// TIA Portal project "Parking_Lort_V15.1" (V15.1)

(* hardware
DEVICE "S7-1200 station_1"  S7-1200 Station
   slot 0: "Rack_0"  S7-1200 Rack  Rack  V1.0
   slot 1: "PLC_1"  CPU 1212C DC/DC/Rly  6ES7 212-1HE40-0XB0  V4.2
*)

// ===== PLC "PLC_1"  CPU 1212C DC/DC/Rly =====

VAR_GLOBAL   // PLC tag table "Default tag table"
   "I_IN barrier is down" AT %I0.0 : Bool;
   "I_IN barrier is up" AT %I0.1 : Bool;
   "I_OUT barrier is down" AT %I0.2 : Bool;
   "I_OUT barrier is up" AT %I0.3 : Bool;
   "I_Car is at the barrier IN" AT %I0.4 : Bool;
   "I_Car is at the barrier OUT" AT %I0.5 : Bool;
   "Q_IN barrier up" AT %Q0.0 : Bool;
   "Q_OUT barrier up" AT %Q0.1 : Bool;
   "Q_Red signal IN" AT %Q0.2 : Bool;
   "Q_Green signal IN" AT %Q0.3 : Bool;
   "Q_Red signal OUT" AT %Q0.4 : Bool;
   "Q_Green signal OUT" AT %Q0.5 : Bool;
END_VAR

DATA_BLOCK "Barrier_DB"   // DB1
{ S7_Optimized_Access := 'TRUE' }
VERSION : 0.1
// stored: InstanceOfName ENTER_Barrier
"ENTER_Barrier"
BEGIN
END_DATA_BLOCK

DATA_BLOCK "EXIT_Barrier_DB"   // DB2
{ S7_Optimized_Access := 'TRUE' }
VERSION : 0.1
// stored: InstanceOfName EXIT_Barrier
"EXIT_Barrier"
BEGIN
END_DATA_BLOCK

FUNCTION_BLOCK "ENTER_Barrier"   // FB1, LAD
TITLE = Barriers
{ S7_Optimized_Access := 'TRUE' }
VERSION : 0.1
BEGIN

REGION Network 1: ENTER
   // Condition to lift up the barrier
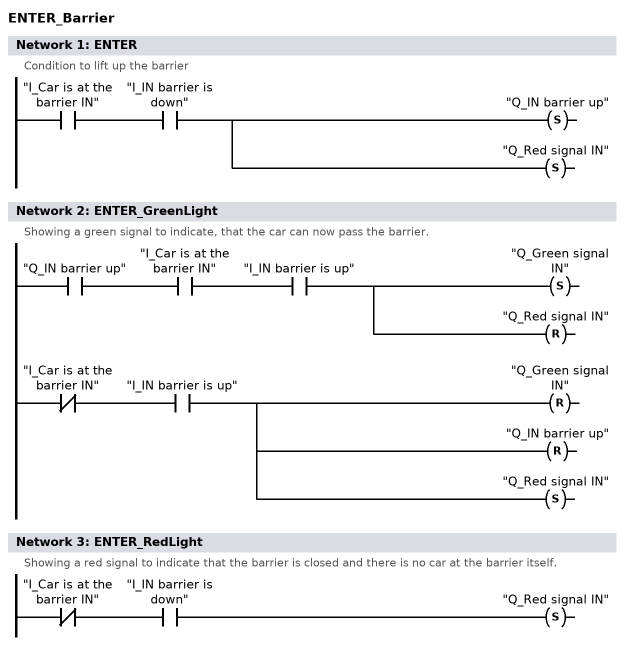
   RUNG wire#powerrail
      Contact( "I_Car is at the barrier IN" )
      Contact( "I_IN barrier is down" )
      wire#w1
      S_Coil( "Q_IN barrier up" )
   END_RUNG
   RUNG wire#w1
      S_Coil( "Q_Red signal IN" )
   END_RUNG
   // the same network as SCL:
   IF "I_Car is at the barrier IN" AND "I_IN barrier is down" THEN
       "Q_IN barrier up" := TRUE;
       "Q_Red signal IN" := TRUE;
   END_IF;
END_REGION

REGION Network 2: ENTER_GreenLight
   // Showing a green signal to indicate, that the car can now pass the barrier.
   RUNG wire#powerrail
      Contact( "Q_IN barrier up" )
      Contact( "I_Car is at the barrier IN" )
      Contact( "I_IN barrier is up" )
      wire#w1
      S_Coil( "Q_Green signal IN" )
   END_RUNG
   RUNG wire#w1
      R_Coil( "Q_Red signal IN" )
   END_RUNG
   RUNG wire#powerrail
      I_Contact( "I_Car is at the barrier IN" )
      Contact( "I_IN barrier is up" )
      wire#w2
      R_Coil( "Q_Green signal IN" )
   END_RUNG
   RUNG wire#w2
      R_Coil( "Q_IN barrier up" )
   END_RUNG
   RUNG wire#w2
      S_Coil( "Q_Red signal IN" )
   END_RUNG
   // the same network as SCL:
   IF "Q_IN barrier up" AND "I_Car is at the barrier IN" AND "I_IN barrier is up" THEN
       "Q_Green signal IN" := TRUE;
       "Q_Red signal IN" := FALSE;
   END_IF;
   IF NOT "I_Car is at the barrier IN" AND "I_IN barrier is up" THEN
       "Q_Green signal IN" := FALSE;
       "Q_IN barrier up" := FALSE;
       "Q_Red signal IN" := TRUE;
   END_IF;
END_REGION

REGION Network 3: ENTER_RedLight
   // Showing a red signal to indicate that the barrier is closed and there is no car at the barrier itself.
   RUNG wire#powerrail
      I_Contact( "I_Car is at the barrier IN" )
      Contact( "I_IN barrier is down" )
      S_Coil( "Q_Red signal IN" )
   END_RUNG
   // the same network as SCL:
   IF NOT "I_Car is at the barrier IN" AND "I_IN barrier is down" THEN "Q_Red signal IN" := TRUE; END_IF;
END_REGION
END_FUNCTION_BLOCK

FUNCTION_BLOCK "EXIT_Barrier"   // FB2, LAD
{ S7_Optimized_Access := 'TRUE' }
VERSION : 0.1
BEGIN

REGION Network 1: ENTER
   // Condition to lift up the barrier
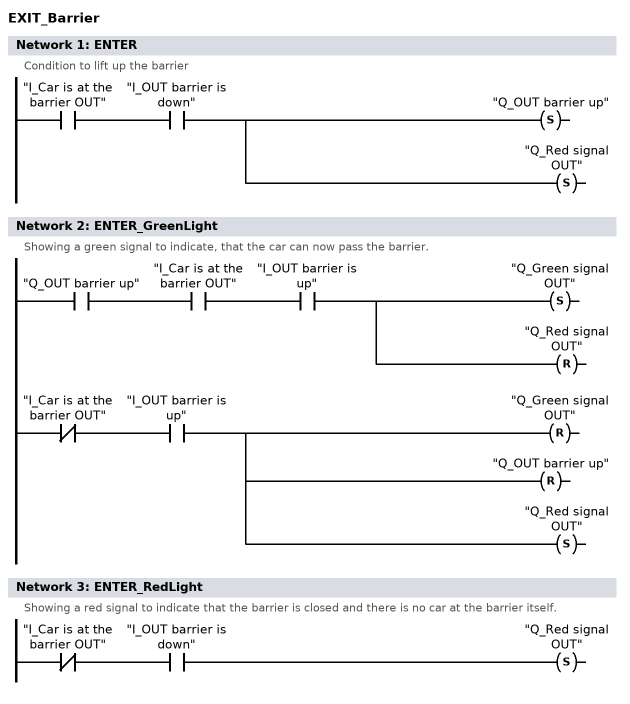
   RUNG wire#powerrail
      Contact( "I_Car is at the barrier OUT" )
      Contact( "I_OUT barrier is down" )
      wire#w1
      S_Coil( "Q_OUT barrier up" )
   END_RUNG
   RUNG wire#w1
      S_Coil( "Q_Red signal OUT" )
   END_RUNG
   // the same network as SCL:
   IF "I_Car is at the barrier OUT" AND "I_OUT barrier is down" THEN
       "Q_OUT barrier up" := TRUE;
       "Q_Red signal OUT" := TRUE;
   END_IF;
END_REGION

REGION Network 2: ENTER_GreenLight
   // Showing a green signal to indicate, that the car can now pass the barrier.
   RUNG wire#powerrail
      Contact( "Q_OUT barrier up" )
      Contact( "I_Car is at the barrier OUT" )
      Contact( "I_OUT barrier is up" )
      wire#w1
      S_Coil( "Q_Green signal OUT" )
   END_RUNG
   RUNG wire#w1
      R_Coil( "Q_Red signal OUT" )
   END_RUNG
   RUNG wire#powerrail
      I_Contact( "I_Car is at the barrier OUT" )
      Contact( "I_OUT barrier is up" )
      wire#w2
      R_Coil( "Q_Green signal OUT" )
   END_RUNG
   RUNG wire#w2
      R_Coil( "Q_OUT barrier up" )
   END_RUNG
   RUNG wire#w2
      S_Coil( "Q_Red signal OUT" )
   END_RUNG
   // the same network as SCL:
   IF "Q_OUT barrier up" AND "I_Car is at the barrier OUT" AND "I_OUT barrier is up" THEN
       "Q_Green signal OUT" := TRUE;
       "Q_Red signal OUT" := FALSE;
   END_IF;
   IF NOT "I_Car is at the barrier OUT" AND "I_OUT barrier is up" THEN
       "Q_Green signal OUT" := FALSE;
       "Q_OUT barrier up" := FALSE;
       "Q_Red signal OUT" := TRUE;
   END_IF;
END_REGION

REGION Network 3: ENTER_RedLight
   // Showing a red signal to indicate that the barrier is closed and there is no car at the barrier itself.
   RUNG wire#powerrail
      I_Contact( "I_Car is at the barrier OUT" )
      Contact( "I_OUT barrier is down" )
      S_Coil( "Q_Red signal OUT" )
   END_RUNG
   // the same network as SCL:
   IF NOT "I_Car is at the barrier OUT" AND "I_OUT barrier is down" THEN "Q_Red signal OUT" := TRUE; END_IF;
END_REGION
END_FUNCTION_BLOCK

ORGANIZATION_BLOCK "Main"   // OB1, LAD, ProgramCycle
TITLE = "Main Program Sweep (Cycle)"
{ S7_Optimized_Access := 'TRUE' }
VERSION : 0.1
   VAR_INPUT
      Initial_Call : Bool;   // Initial call of this OB
      Remanence : Bool;   // =True, if remanent data are available
   END_VAR
BEGIN

REGION Network 1
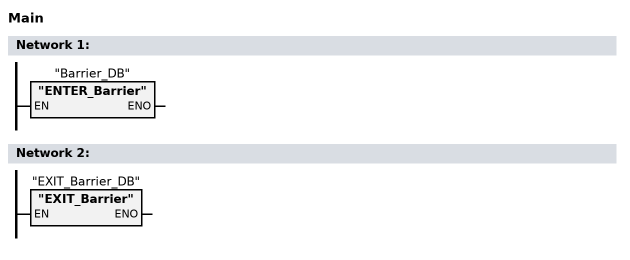
   RUNG wire#powerrail
      "Barrier_DB"()
   END_RUNG
   // the same network as SCL:
   "Barrier_DB"();   // "ENTER_Barrier"
END_REGION

REGION Network 2
   RUNG wire#powerrail
      "EXIT_Barrier_DB"()
   END_RUNG
   // the same network as SCL:
   "EXIT_Barrier_DB"();   // "EXIT_Barrier"
END_REGION
END_ORGANIZATION_BLOCK